{attribute 'qualified_only'}
TYPE E_SafetyGroup_Diag : (
		NoError		  := 0,
		FbError		  := 1,
		ComError	  := 2,
		ModuleError	  := 3,
		CmpError	  := 4,
		DeactiveError := 5,
		RestartError  := 6
	) UINT;
END_TYPE

(* stored: Version 1.1.0.1, ProductVersion 3.1.4026.18
   DUT E_SafetyGroup_Diag: Id {cd4fab5e-cd39-0c18-3fe0-daf642f4834c} *)
